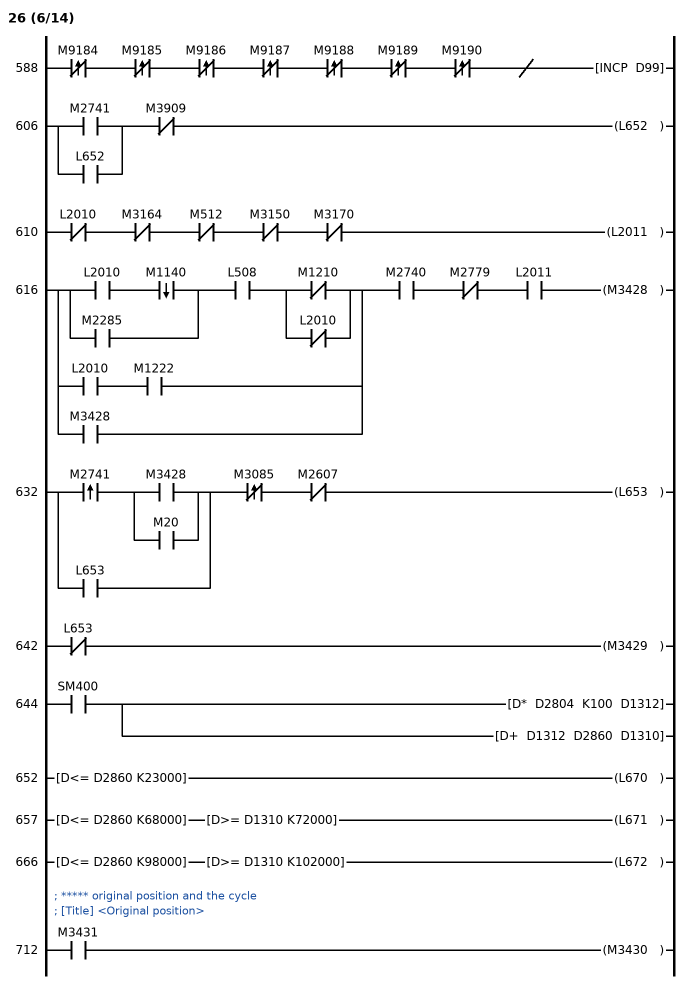
588   LDPI    M9184
      ANDPI   M9185
      ANDPI   M9186
      ANDPI   M9187
      ANDPI   M9188
      ANDPI   M9189
      ANDPI   M9190
      INV
      INCP    D99
606   LD      M2741
      OR      L652
      ANI     M3909
      OUT     L652
610   LDI     L2010
      ANI     M3164
      ANI     M512
      ANI     M3150
      ANI     M3170
      OUT     L2011
616   LD      L2010
      ANDF    M1140
      OR      M2285
      AND     L508
      LDI     M1210
      ORI     L2010
      ANB
      LD      L2010
      AND     M1222
      ORB
      OR      M3428
      AND     M2740
      ANI     M2779
      AND     L2011
      OUT     M3428
632   LDP     M2741
      LD      M3428
      OR      M20
      ANB
      OR      L653
      ANDPI   M3085
      ANI     M2607
      OUT     L653
642   LDI     L653
      OUT     M3429
644   LD      SM400
      D*      D2804 K100 D1312
      D+      D1312 D2860 D1310
652   LDD<=   D2860 K23000
      OUT     L670
657   LDD<=   D2860 K68000
      ANDD>=  D1310 K72000
      OUT     L671
666   LDD<=   D2860 K98000
      ANDD>=  D1310 K102000
      OUT     L672
; ***** original position and the cycle
; [Title] <Original position>
712   LD      M3431
      OUT     M3430
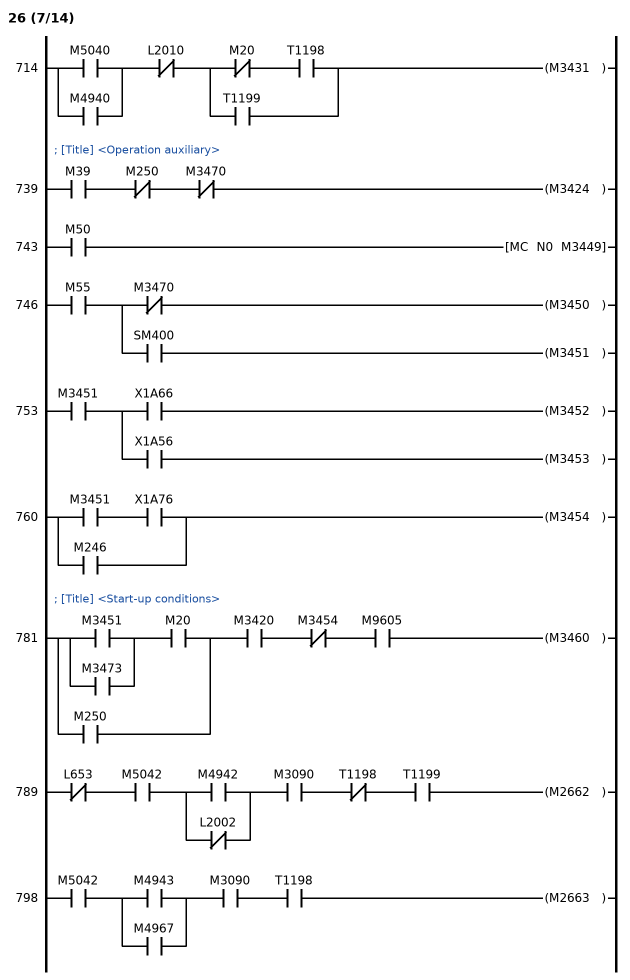
714   LD      M5040
      OR      M4940
      ANI     L2010
      LDI     M20
      AND     T1198
      OR      T1199
      ANB
      OUT     M3431
; [Title] <Operation auxiliary>
739   LD      M39
      ANI     M250
      ANI     M3470
      OUT     M3424
743   LD      M50
      MC      N0 M3449
746   LD      M55
      MPS
      ANI     M3470
      OUT     M3450
      MPP
      AND     SM400
      OUT     M3451
753   LD      M3451
      MPS
      AND     X1A66
      OUT     M3452
      MPP
      AND     X1A56
      OUT     M3453
760   LD      M3451
      AND     X1A76
      OR      M246
      OUT     M3454
; [Title] <Start-up conditions>
781   LD      M3451
      OR      M3473
      AND     M20
      OR      M250
      AND     M3420
      ANI     M3454
      AND     M9605
      OUT     M3460
789   LDI     L653
      AND     M5042
      LD      M4942
      ORI     L2002
      ANB
      AND     M3090
      ANI     T1198
      AND     T1199
      OUT     M2662
798   LD      M5042
      LD      M4943
      OR      M4967
      ANB
      AND     M3090
      AND     T1198
      OUT     M2663
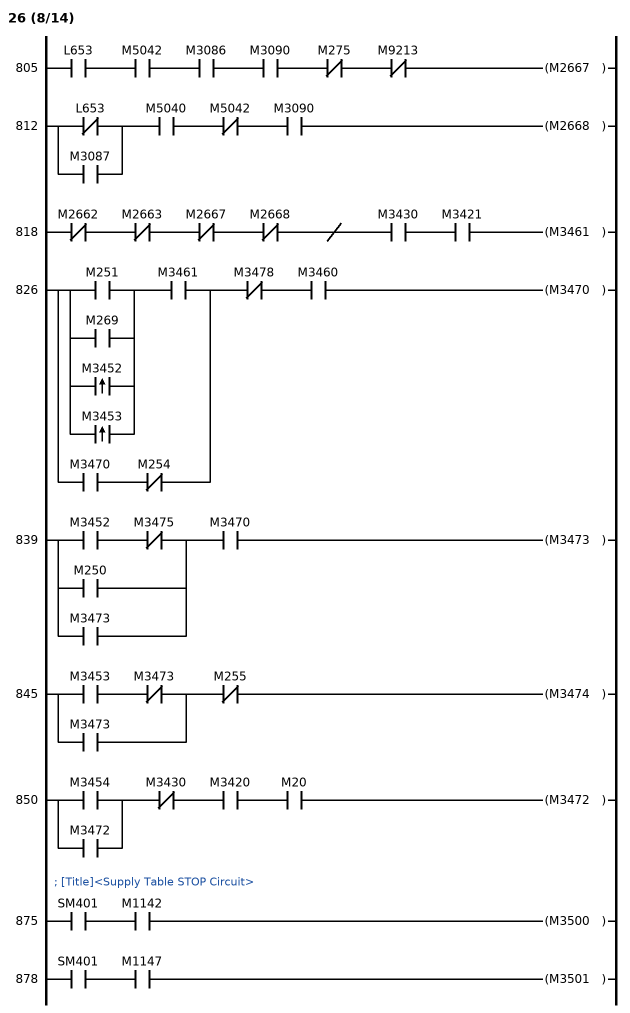
805   LD      L653
      AND     M5042
      AND     M3086
      AND     M3090
      ANI     M275
      ANI     M9213
      OUT     M2667
812   LDI     L653
      OR      M3087
      AND     M5040
      ANI     M5042
      AND     M3090
      OUT     M2668
818   LDI     M2662
      ANI     M2663
      ANI     M2667
      ANI     M2668
      INV
      AND     M3430
      AND     M3421
      OUT     M3461
826   LD      M251
      OR      M269
      ORP     M3452
      ORP     M3453
      AND     M3461
      LD      M3470
      ANI     M254
      ORB
      ANI     M3478
      AND     M3460
      OUT     M3470
839   LD      M3452
      ANI     M3475
      OR      M250
      OR      M3473
      AND     M3470
      OUT     M3473
845   LD      M3453
      ANI     M3473
      OR      M3473
      ANI     M255
      OUT     M3474
850   LD      M3454
      OR      M3472
      ANI     M3430
      AND     M3420
      AND     M20
      OUT     M3472
; [Title]<Supply Table STOP Circuit>
875   LD      SM401
      AND     M1142
      OUT     M3500
878   LD      SM401
      AND     M1147
      OUT     M3501
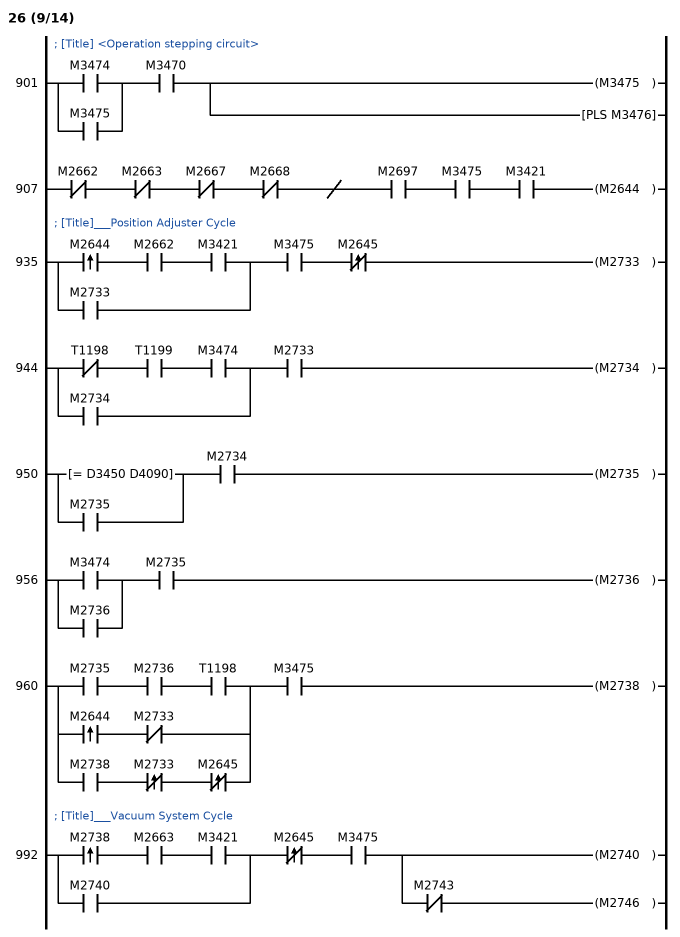
; [Title] <Operation stepping circuit>
901   LD      M3474
      OR      M3475
      AND     M3470
      OUT     M3475
      PLS     M3476
907   LDI     M2662
      ANI     M2663
      ANI     M2667
      ANI     M2668
      INV
      AND     M2697
      AND     M3475
      AND     M3421
      OUT     M2644
; [Title]___Position Adjuster Cycle
935   LDP     M2644
      AND     M2662
      AND     M3421
      OR      M2733
      AND     M3475
      ANDPI   M2645
      OUT     M2733
944   LDI     T1198
      AND     T1199
      AND     M3474
      OR      M2734
      AND     M2733
      OUT     M2734
950   LD=     D3450 D4090
      OR      M2735
      AND     M2734
      OUT     M2735
956   LD      M3474
      OR      M2736
      AND     M2735
      OUT     M2736
960   LD      M2735
      AND     M2736
      AND     T1198
      LDP     M2644
      ANI     M2733
      ORB
      LD      M2738
      ANDPI   M2733
      ANDPI   M2645
      ORB
      AND     M3475
      OUT     M2738
; [Title]___Vacuum System Cycle
992   LDP     M2738
      AND     M2663
      AND     M3421
      OR      M2740
      ANDPI   M2645
      AND     M3475
      OUT     M2740
      ANI     M2743
      OUT     M2746
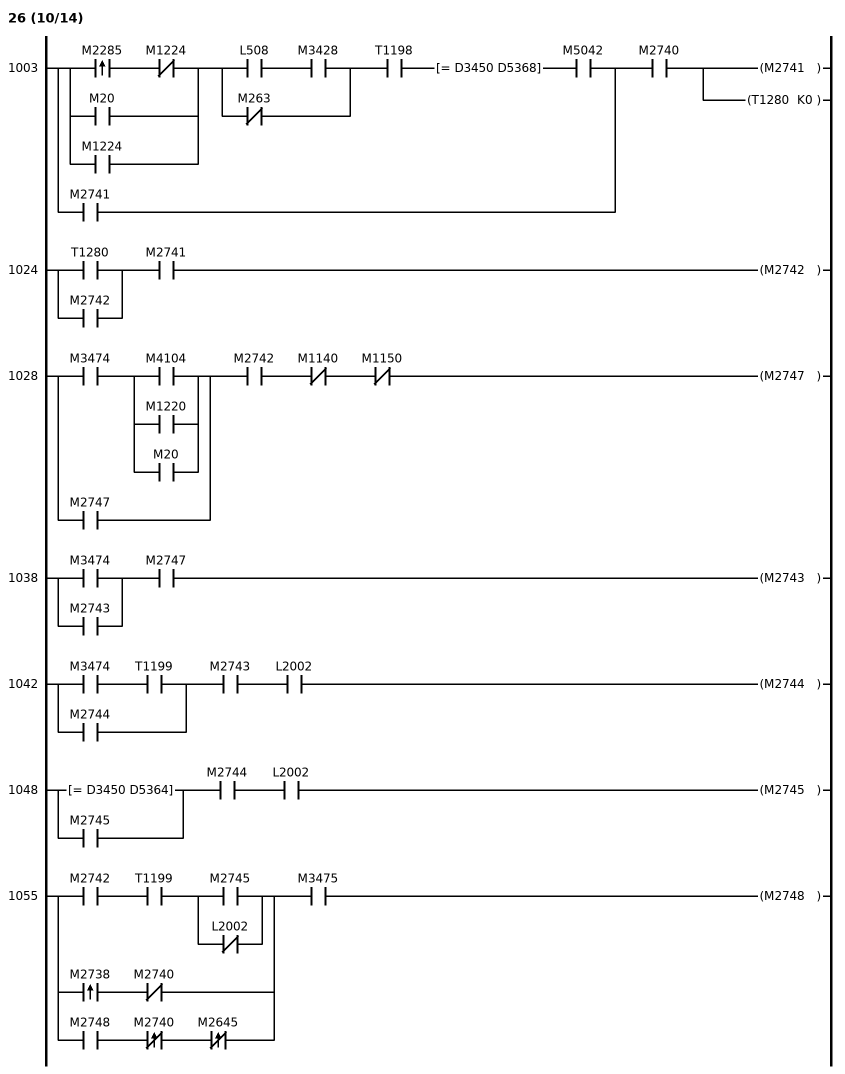
1003  LDP     M2285
      ANI     M1224
      OR      M20
      OR      M1224
      LD      L508
      AND     M3428
      ORI     M263
      ANB
      AND     T1198
      AND=    D3450 D5368
      AND     M5042
      OR      M2741
      AND     M2740
      OUT     M2741
      OUT     T1280 K0
1024  LD      T1280
      OR      M2742
      AND     M2741
      OUT     M2742
1028  LD      M3474
      LD      M4104
      OR      M1220
      OR      M20
      ANB
      OR      M2747
      AND     M2742
      ANI     M1140
      ANI     M1150
      OUT     M2747
1038  LD      M3474
      OR      M2743
      AND     M2747
      OUT     M2743
1042  LD      M3474
      AND     T1199
      OR      M2744
      AND     M2743
      AND     L2002
      OUT     M2744
1048  LD=     D3450 D5364
      OR      M2745
      AND     M2744
      AND     L2002
      OUT     M2745
1055  LD      M2742
      AND     T1199
      LD      M2745
      ORI     L2002
      ANB
      LDP     M2738
      ANI     M2740
      ORB
      LD      M2748
      ANDPI   M2740
      ANDPI   M2645
      ORB
      AND     M3475
      OUT     M2748
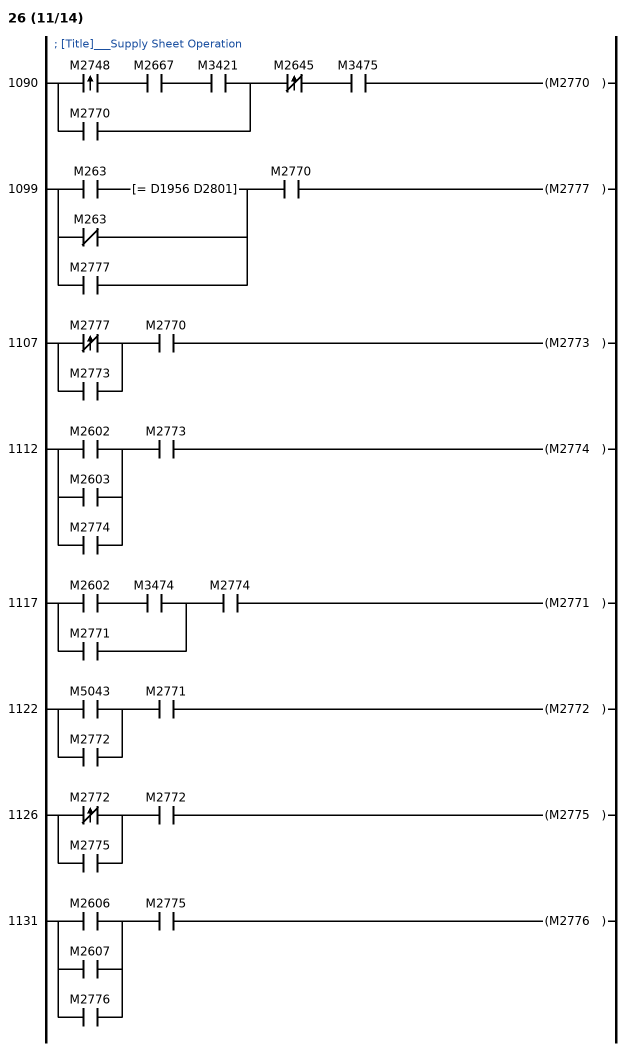
; [Title]___Supply Sheet Operation
1090  LDP     M2748
      AND     M2667
      AND     M3421
      OR      M2770
      ANDPI   M2645
      AND     M3475
      OUT     M2770
1099  LD      M263
      AND=    D1956 D2801
      ORI     M263
      OR      M2777
      AND     M2770
      OUT     M2777
1107  LDPI    M2777
      OR      M2773
      AND     M2770
      OUT     M2773
1112  LD      M2602
      OR      M2603
      OR      M2774
      AND     M2773
      OUT     M2774
1117  LD      M2602
      AND     M3474
      OR      M2771
      AND     M2774
      OUT     M2771
1122  LD      M5043
      OR      M2772
      AND     M2771
      OUT     M2772
1126  LDPI    M2772
      OR      M2775
      AND     M2772
      OUT     M2775
1131  LD      M2606
      OR      M2607
      OR      M2776
      AND     M2775
      OUT     M2776
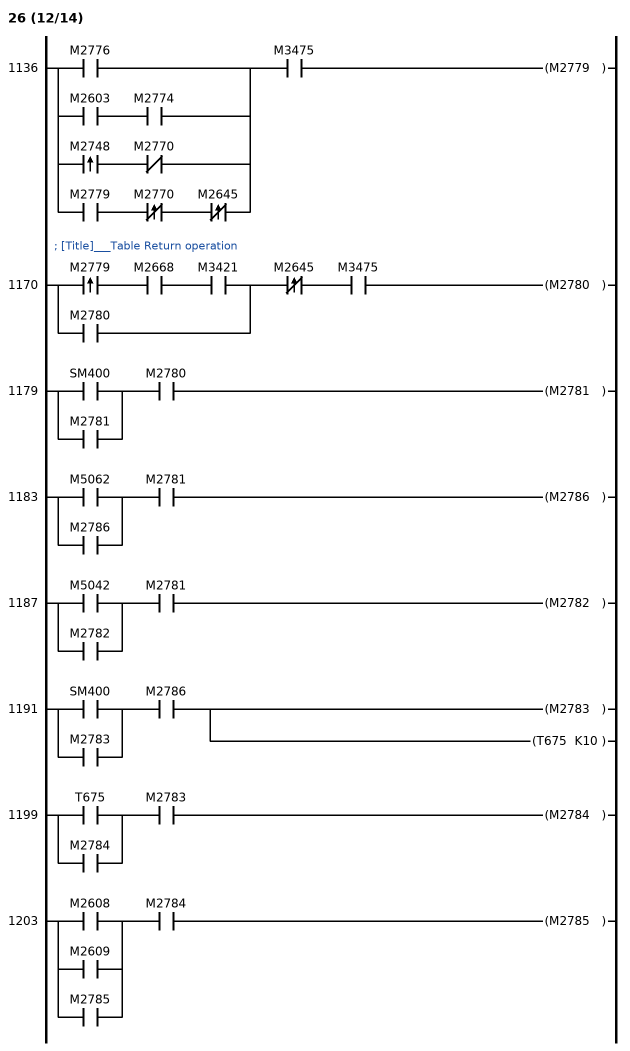
1136  LD      M2776
      LD      M2603
      AND     M2774
      ORB
      LDP     M2748
      ANI     M2770
      ORB
      LD      M2779
      ANDPI   M2770
      ANDPI   M2645
      ORB
      AND     M3475
      OUT     M2779
; [Title]___Table Return operation
1170  LDP     M2779
      AND     M2668
      AND     M3421
      OR      M2780
      ANDPI   M2645
      AND     M3475
      OUT     M2780
1179  LD      SM400
      OR      M2781
      AND     M2780
      OUT     M2781
1183  LD      M5062
      OR      M2786
      AND     M2781
      OUT     M2786
1187  LD      M5042
      OR      M2782
      AND     M2781
      OUT     M2782
1191  LD      SM400
      OR      M2783
      AND     M2786
      OUT     M2783
      OUT     T675 K10
1199  LD      T675
      OR      M2784
      AND     M2783
      OUT     M2784
1203  LD      M2608
      OR      M2609
      OR      M2785
      AND     M2784
      OUT     M2785
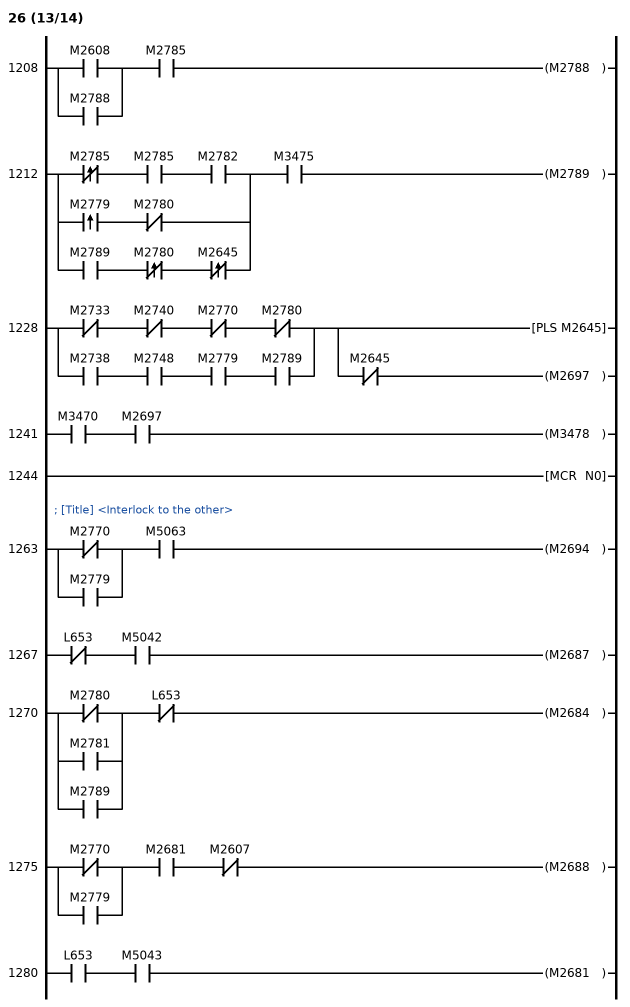
1208  LD      M2608
      OR      M2788
      AND     M2785
      OUT     M2788
1212  LDPI    M2785
      AND     M2785
      AND     M2782
      LDP     M2779
      ANI     M2780
      ORB
      LD      M2789
      ANDPI   M2780
      ANDPI   M2645
      ORB
      AND     M3475
      OUT     M2789
1228  LDI     M2733
      ANI     M2740
      ANI     M2770
      ANI     M2780
      LD      M2738
      AND     M2748
      AND     M2779
      AND     M2789
      ORB
      PLS     M2645
      ANI     M2645
      OUT     M2697
1241  LD      M3470
      AND     M2697
      OUT     M3478
1244  MCR     N0
; [Title] <Interlock to the other>
1263  LDI     M2770
      OR      M2779
      AND     M5063
      OUT     M2694
1267  LDI     L653
      AND     M5042
      OUT     M2687
1270  LDI     M2780
      OR      M2781
      OR      M2789
      ANI     L653
      OUT     M2684
1275  LDI     M2770
      OR      M2779
      AND     M2681
      ANI     M2607
      OUT     M2688
1280  LD      L653
      AND     M5043
      OUT     M2681
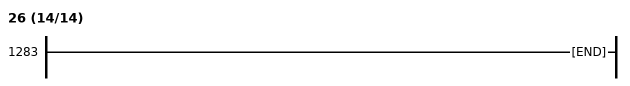
1283  END
END_PROGRAM

PROGRAM 70
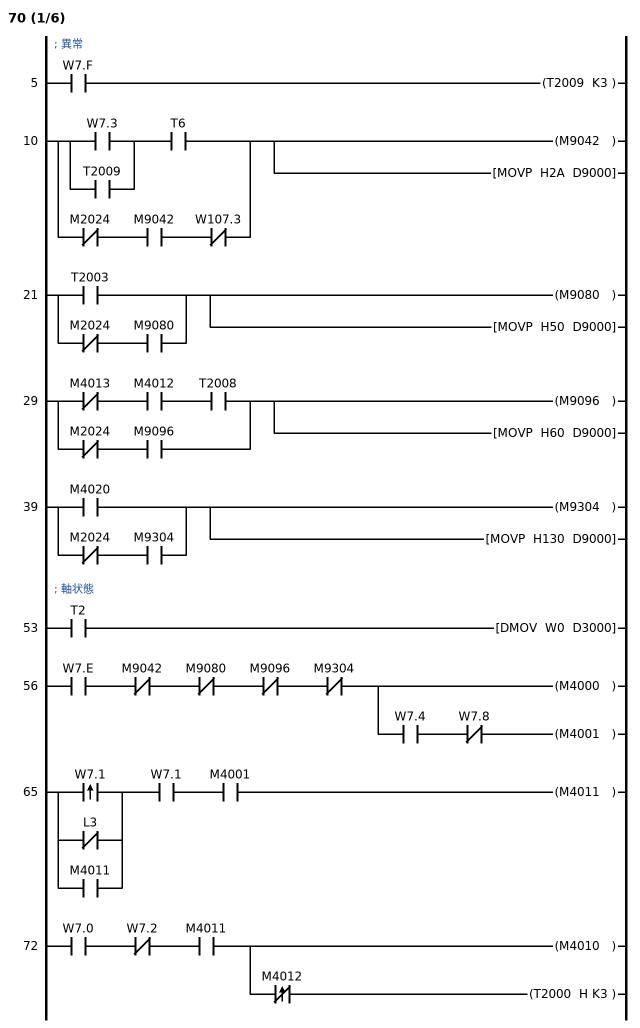
; 異常
5     LD      W7.F
      OUT     T2009 K3
10    LD      W7.3
      OR      T2009
      AND     T6
      LDI     M2024
      AND     M9042
      ANI     W107.3
      ORB
      OUT     M9042
      MOVP    H2A D9000
21    LD      T2003
      LDI     M2024
      AND     M9080
      ORB
      OUT     M9080
      MOVP    H50 D9000
29    LDI     M4013
      AND     M4012
      AND     T2008
      LDI     M2024
      AND     M9096
      ORB
      OUT     M9096
      MOVP    H60 D9000
39    LD      M4020
      LDI     M2024
      AND     M9304
      ORB
      OUT     M9304
      MOVP    H130 D9000
; 軸状態
53    LD      T2
      DMOV    W0 D3000
56    LD      W7.E
      ANI     M9042
      ANI     M9080
      ANI     M9096
      ANI     M9304
      OUT     M4000
      AND     W7.4
      ANI     W7.8
      OUT     M4001
65    LDP     W7.1
      ORI     L3
      OR      M4011
      AND     W7.1
      AND     M4001
      OUT     M4011
72    LD      W7.0
      ANI     W7.2
      AND     M4011
      OUT     M4010
      ANDPI   M4012
      OUTH    T2000 K3
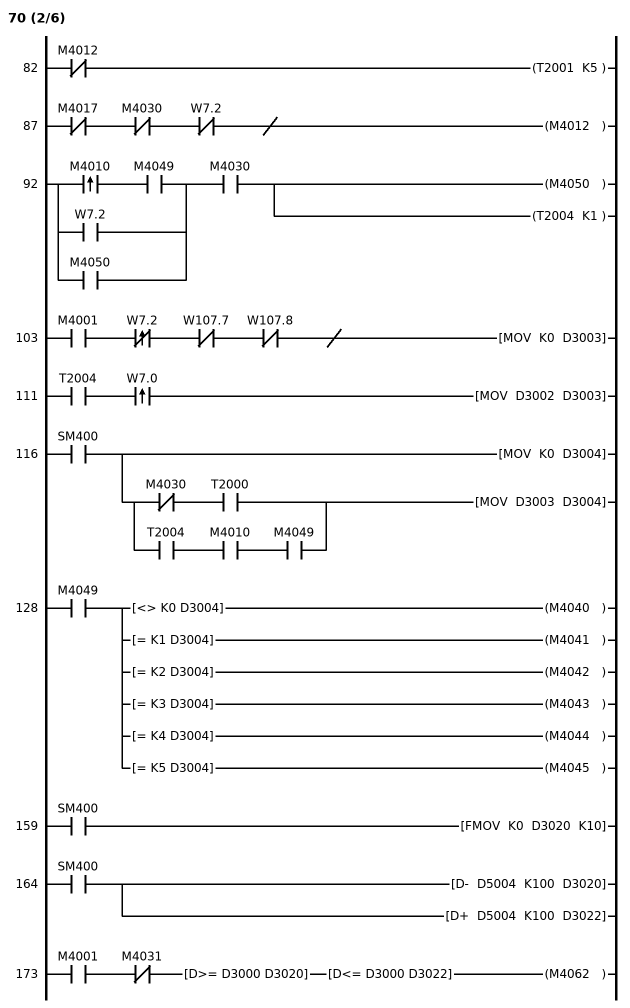
82    LDI     M4012
      OUT     T2001 K5
87    LDI     M4017
      ANI     M4030
      ANI     W7.2
      INV
      OUT     M4012
92    LDP     M4010
      AND     M4049
      OR      W7.2
      OR      M4050
      AND     M4030
      OUT     M4050
      OUT     T2004 K1
103   LD      M4001
      ANDPI   W7.2
      ANI     W107.7
      ANI     W107.8
      INV
      MOV     K0 D3003
111   LD      T2004
      ANDP    W7.0
      MOV     D3002 D3003
116   LD      SM400
      MOV     K0 D3004
      LDI     M4030
      AND     T2000
      LD      T2004
      AND     M4010
      AND     M4049
      ORB
      ANB
      MOV     D3003 D3004
128   LD      M4049
      MPS
      AND<>   K0 D3004
      OUT     M4040
      MRD
      AND=    K1 D3004
      OUT     M4041
      MRD
      AND=    K2 D3004
      OUT     M4042
      MRD
      AND=    K3 D3004
      OUT     M4043
      MRD
      AND=    K4 D3004
      OUT     M4044
      MPP
      AND=    K5 D3004
      OUT     M4045
159   LD      SM400
      FMOV    K0 D3020 K10
164   LD      SM400
      D-      D5004 K100 D3020
      D+      D5004 K100 D3022
173   LD      M4001
      ANI     M4031
      ANDD>=  D3000 D3020
      ANDD<=  D3000 D3022
      OUT     M4062
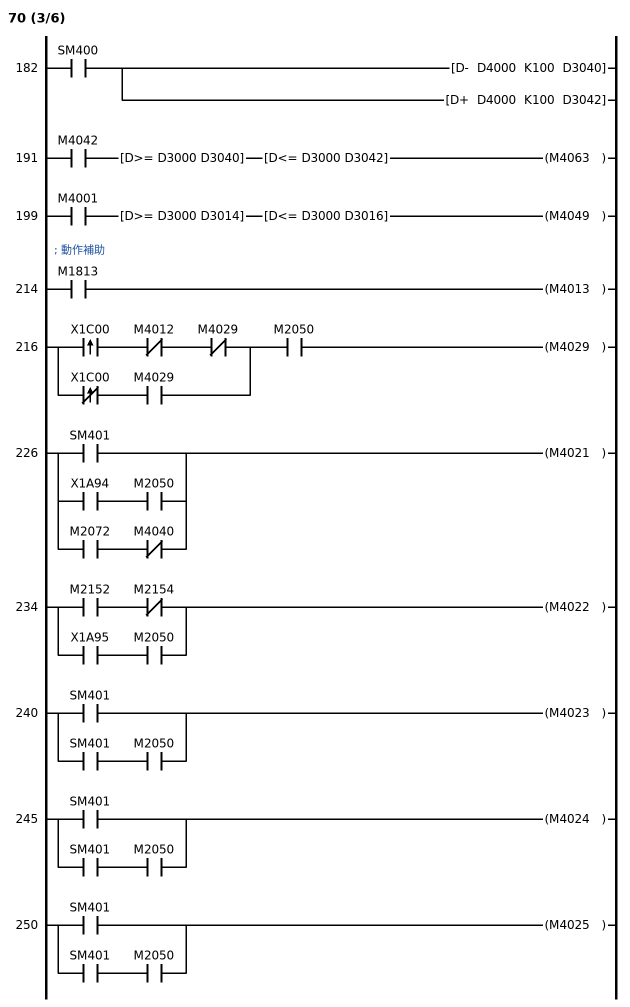
182   LD      SM400
      D-      D4000 K100 D3040
      D+      D4000 K100 D3042
191   LD      M4042
      ANDD>=  D3000 D3040
      ANDD<=  D3000 D3042
      OUT     M4063
199   LD      M4001
      ANDD>=  D3000 D3014
      ANDD<=  D3000 D3016
      OUT     M4049
; 動作補助
214   LD      M1813
      OUT     M4013
216   LDP     X1C00
      ANI     M4012
      ANI     M4029
      LDPI    X1C00
      AND     M4029
      ORB
      AND     M2050
      OUT     M4029
226   LD      SM401
      LD      X1A94
      AND     M2050
      ORB
      LD      M2072
      ANI     M4040
      ORB
      OUT     M4021
234   LD      M2152
      ANI     M2154
      LD      X1A95
      AND     M2050
      ORB
      OUT     M4022
240   LD      SM401
      LD      SM401
      AND     M2050
      ORB
      OUT     M4023
245   LD      SM401
      LD      SM401
      AND     M2050
      ORB
      OUT     M4024
250   LD      SM401
      LD      SM401
      AND     M2050
      ORB
      OUT     M4025
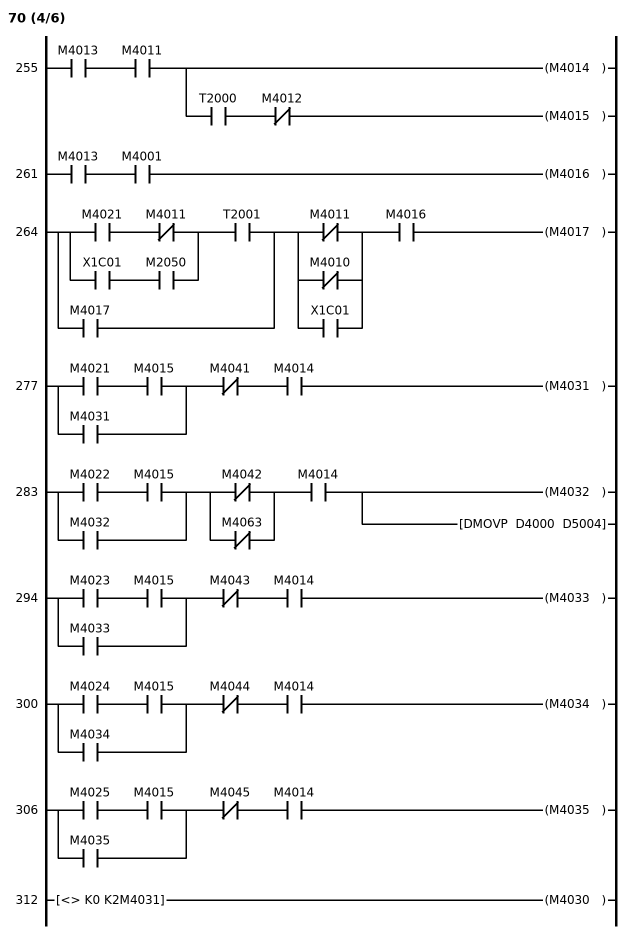
255   LD      M4013
      AND     M4011
      OUT     M4014
      AND     T2000
      ANI     M4012
      OUT     M4015
261   LD      M4013
      AND     M4001
      OUT     M4016
264   LD      M4021
      ANI     M4011
      LD      X1C01
      AND     M2050
      ORB
      AND     T2001
      OR      M4017
      LDI     M4011
      ORI     M4010
      OR      X1C01
      ANB
      AND     M4016
      OUT     M4017
277   LD      M4021
      AND     M4015
      OR      M4031
      ANI     M4041
      AND     M4014
      OUT     M4031
283   LD      M4022
      AND     M4015
      OR      M4032
      LDI     M4042
      ORI     M4063
      ANB
      AND     M4014
      OUT     M4032
      DMOVP   D4000 D5004
294   LD      M4023
      AND     M4015
      OR      M4033
      ANI     M4043
      AND     M4014
      OUT     M4033
300   LD      M4024
      AND     M4015
      OR      M4034
      ANI     M4044
      AND     M4014
      OUT     M4034
306   LD      M4025
      AND     M4015
      OR      M4035
      ANI     M4045
      AND     M4014
      OUT     M4035
312   LD<>    K0 K2M4031
      OUT     M4030
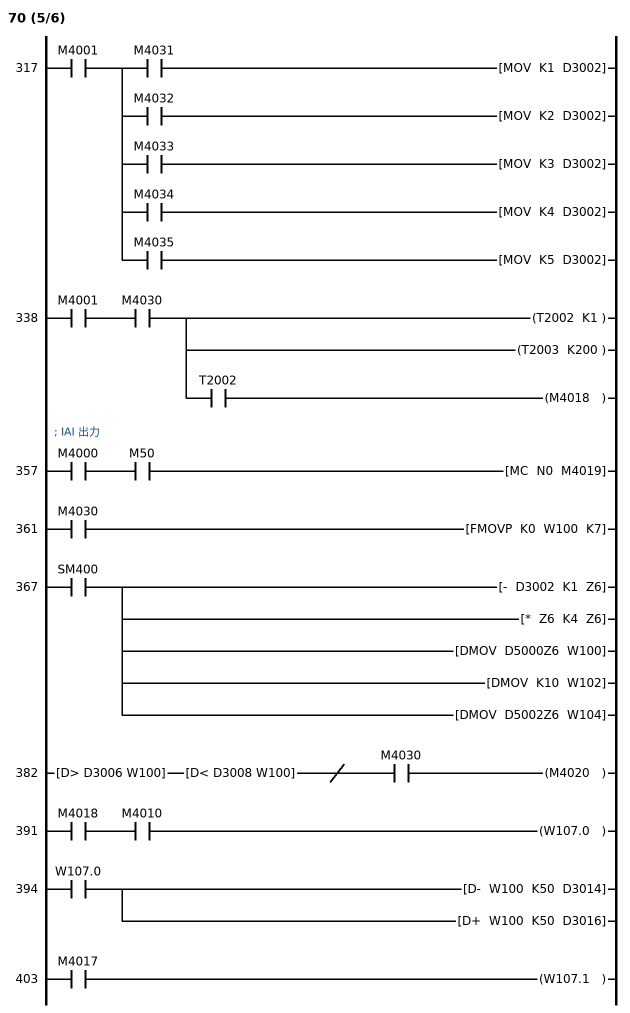
317   LD      M4001
      MPS
      AND     M4031
      MOV     K1 D3002
      MRD
      AND     M4032
      MOV     K2 D3002
      MRD
      AND     M4033
      MOV     K3 D3002
      MRD
      AND     M4034
      MOV     K4 D3002
      MPP
      AND     M4035
      MOV     K5 D3002
338   LD      M4001
      AND     M4030
      OUT     T2002 K1
      OUT     T2003 K200
      AND     T2002
      OUT     M4018
; IAI 出力
357   LD      M4000
      AND     M50
      MC      N0 M4019
361   LD      M4030
      FMOVP   K0 W100 K7
367   LD      SM400
      -       D3002 K1 Z6
      *       Z6 K4 Z6
      DMOV    D5000Z6 W100
      DMOV    K10 W102
      DMOV    D5002Z6 W104
382   LDD>    D3006 W100
      ANDD<   D3008 W100
      INV
      AND     M4030
      OUT     M4020
391   LD      M4018
      AND     M4010
      OUT     W107.0
394   LD      W107.0
      D-      W100 K50 D3014
      D+      W100 K50 D3016
403   LD      M4017
      OUT     W107.1
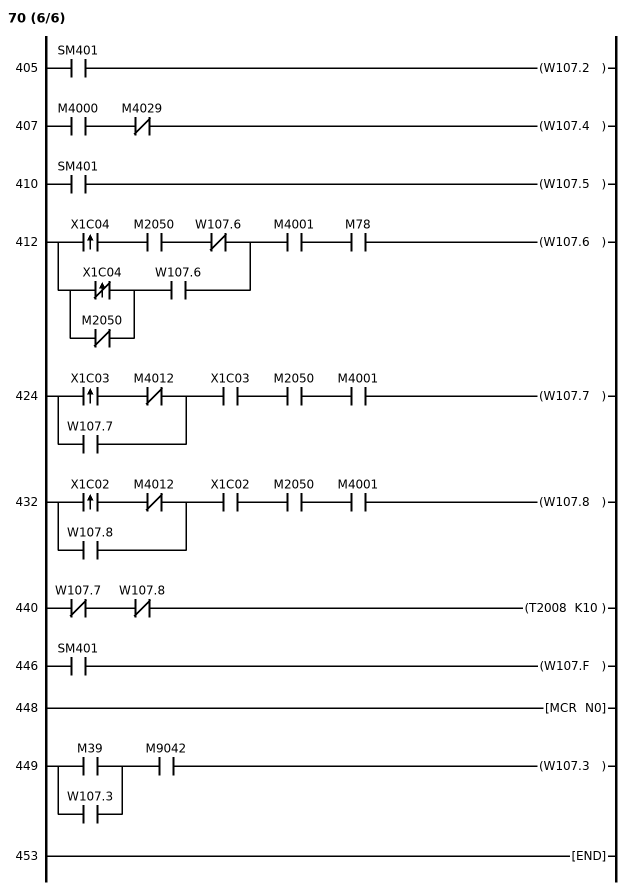
405   LD      SM401
      OUT     W107.2
407   LD      M4000
      ANI     M4029
      OUT     W107.4
410   LD      SM401
      OUT     W107.5
412   LDP     X1C04
      AND     M2050
      ANI     W107.6
      LDPI    X1C04
      ORI     M2050
      AND     W107.6
      ORB
      AND     M4001
      AND     M78
      OUT     W107.6
424   LDP     X1C03
      ANI     M4012
      OR      W107.7
      AND     X1C03
      AND     M2050
      AND     M4001
      OUT     W107.7
432   LDP     X1C02
      ANI     M4012
      OR      W107.8
      AND     X1C02
      AND     M2050
      AND     M4001
      OUT     W107.8
440   LDI     W107.7
      ANI     W107.8
      OUT     T2008 K10
446   LD      SM401
      OUT     W107.F
448   MCR     N0
449   LD      M39
      OR      W107.3
      AND     M9042
      OUT     W107.3
453   END
END_PROGRAM

PROGRAM 71
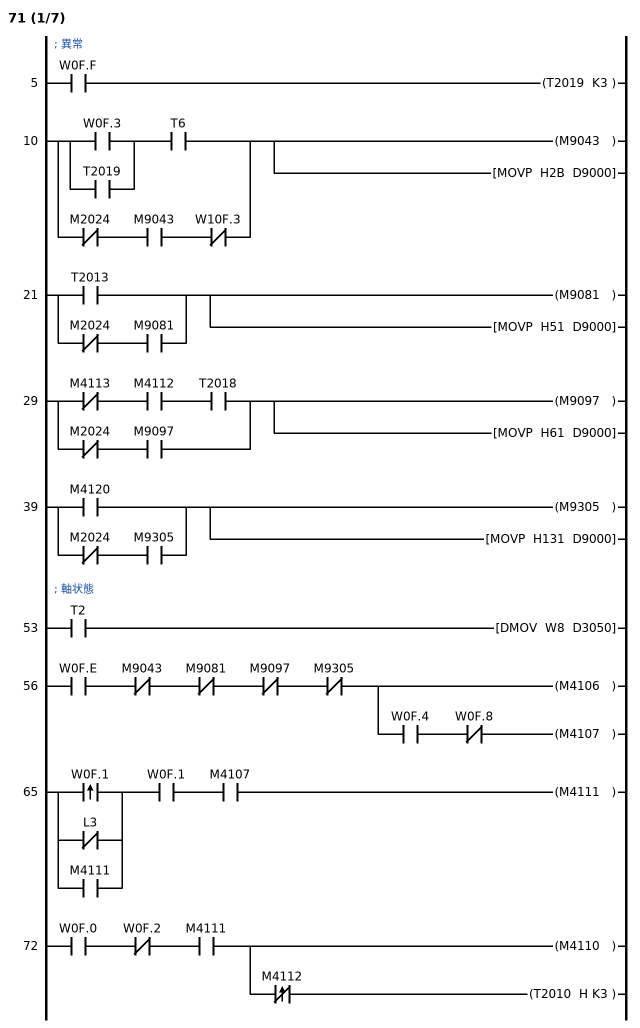
; 異常
5     LD      W0F.F
      OUT     T2019 K3
10    LD      W0F.3
      OR      T2019
      AND     T6
      LDI     M2024
      AND     M9043
      ANI     W10F.3
      ORB
      OUT     M9043
      MOVP    H2B D9000
21    LD      T2013
      LDI     M2024
      AND     M9081
      ORB
      OUT     M9081
      MOVP    H51 D9000
29    LDI     M4113
      AND     M4112
      AND     T2018
      LDI     M2024
      AND     M9097
      ORB
      OUT     M9097
      MOVP    H61 D9000
39    LD      M4120
      LDI     M2024
      AND     M9305
      ORB
      OUT     M9305
      MOVP    H131 D9000
; 軸状態
53    LD      T2
      DMOV    W8 D3050
56    LD      W0F.E
      ANI     M9043
      ANI     M9081
      ANI     M9097
      ANI     M9305
      OUT     M4106
      AND     W0F.4
      ANI     W0F.8
      OUT     M4107
65    LDP     W0F.1
      ORI     L3
      OR      M4111
      AND     W0F.1
      AND     M4107
      OUT     M4111
72    LD      W0F.0
      ANI     W0F.2
      AND     M4111
      OUT     M4110
      ANDPI   M4112
      OUTH    T2010 K3
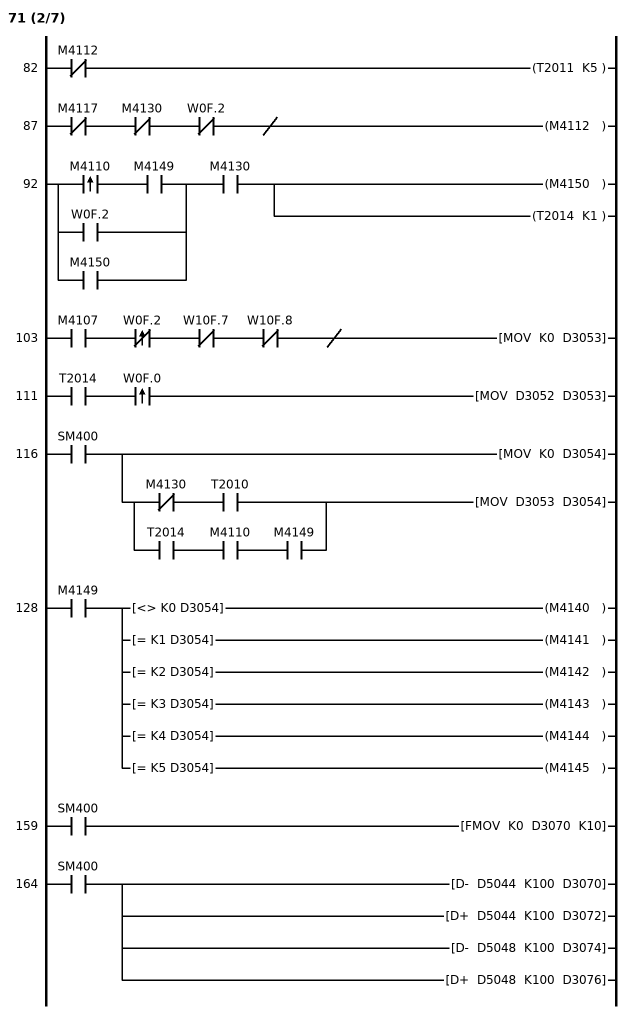
82    LDI     M4112
      OUT     T2011 K5
87    LDI     M4117
      ANI     M4130
      ANI     W0F.2
      INV
      OUT     M4112
92    LDP     M4110
      AND     M4149
      OR      W0F.2
      OR      M4150
      AND     M4130
      OUT     M4150
      OUT     T2014 K1
103   LD      M4107
      ANDPI   W0F.2
      ANI     W10F.7
      ANI     W10F.8
      INV
      MOV     K0 D3053
111   LD      T2014
      ANDP    W0F.0
      MOV     D3052 D3053
116   LD      SM400
      MOV     K0 D3054
      LDI     M4130
      AND     T2010
      LD      T2014
      AND     M4110
      AND     M4149
      ORB
      ANB
      MOV     D3053 D3054
128   LD      M4149
      MPS
      AND<>   K0 D3054
      OUT     M4140
      MRD
      AND=    K1 D3054
      OUT     M4141
      MRD
      AND=    K2 D3054
      OUT     M4142
      MRD
      AND=    K3 D3054
      OUT     M4143
      MRD
      AND=    K4 D3054
      OUT     M4144
      MPP
      AND=    K5 D3054
      OUT     M4145
159   LD      SM400
      FMOV    K0 D3070 K10
164   LD      SM400
      D-      D5044 K100 D3070
      D+      D5044 K100 D3072
      D-      D5048 K100 D3074
      D+      D5048 K100 D3076
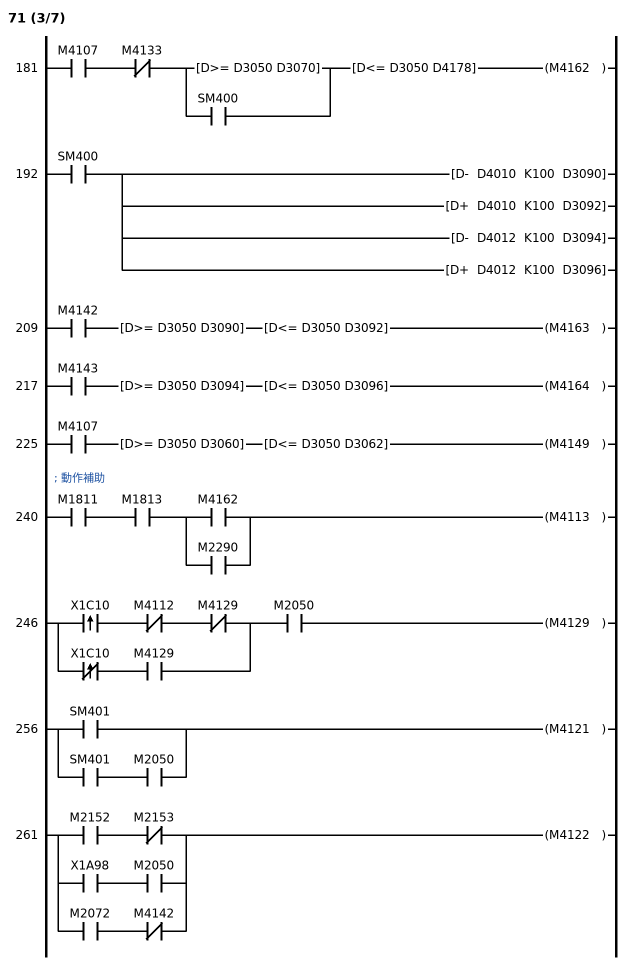
181   LD      M4107
      ANI     M4133
      LDD>=   D3050 D3070
      OR      SM400
      ANB
      ANDD<=  D3050 D4178
      OUT     M4162
192   LD      SM400
      D-      D4010 K100 D3090
      D+      D4010 K100 D3092
      D-      D4012 K100 D3094
      D+      D4012 K100 D3096
209   LD      M4142
      ANDD>=  D3050 D3090
      ANDD<=  D3050 D3092
      OUT     M4163
217   LD      M4143
      ANDD>=  D3050 D3094
      ANDD<=  D3050 D3096
      OUT     M4164
225   LD      M4107
      ANDD>=  D3050 D3060
      ANDD<=  D3050 D3062
      OUT     M4149
; 動作補助
240   LD      M1811
      AND     M1813
      LD      M4162
      OR      M2290
      ANB
      OUT     M4113
246   LDP     X1C10
      ANI     M4112
      ANI     M4129
      LDPI    X1C10
      AND     M4129
      ORB
      AND     M2050
      OUT     M4129
256   LD      SM401
      LD      SM401
      AND     M2050
      ORB
      OUT     M4121
261   LD      M2152
      ANI     M2153
      LD      X1A98
      AND     M2050
      ORB
      LD      M2072
      ANI     M4142
      ORB
      OUT     M4122
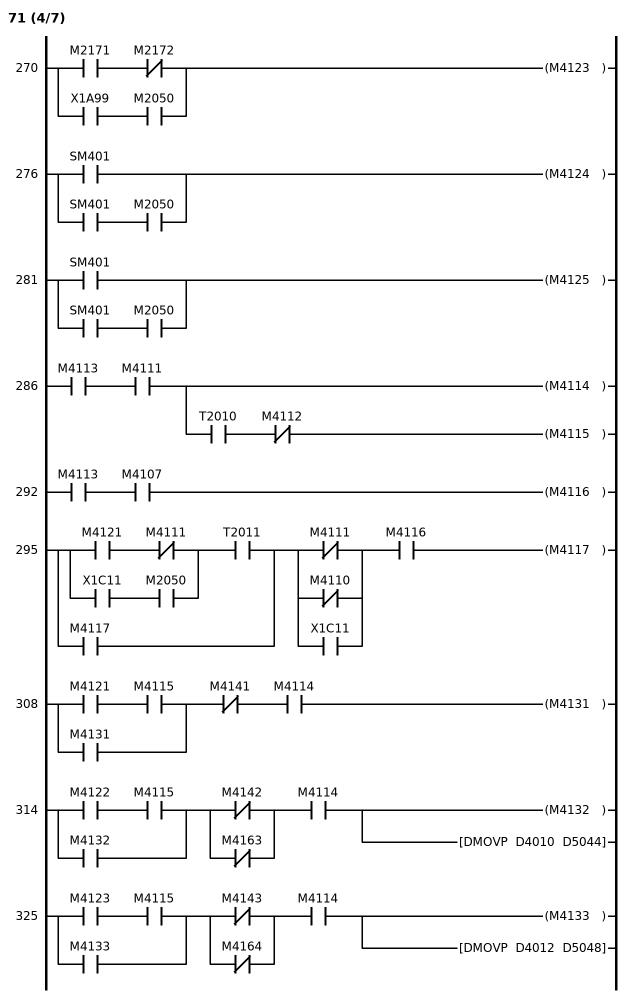
270   LD      M2171
      ANI     M2172
      LD      X1A99
      AND     M2050
      ORB
      OUT     M4123
276   LD      SM401
      LD      SM401
      AND     M2050
      ORB
      OUT     M4124
281   LD      SM401
      LD      SM401
      AND     M2050
      ORB
      OUT     M4125
286   LD      M4113
      AND     M4111
      OUT     M4114
      AND     T2010
      ANI     M4112
      OUT     M4115
292   LD      M4113
      AND     M4107
      OUT     M4116
295   LD      M4121
      ANI     M4111
      LD      X1C11
      AND     M2050
      ORB
      AND     T2011
      OR      M4117
      LDI     M4111
      ORI     M4110
      OR      X1C11
      ANB
      AND     M4116
      OUT     M4117
308   LD      M4121
      AND     M4115
      OR      M4131
      ANI     M4141
      AND     M4114
      OUT     M4131
314   LD      M4122
      AND     M4115
      OR      M4132
      LDI     M4142
      ORI     M4163
      ANB
      AND     M4114
      OUT     M4132
      DMOVP   D4010 D5044
325   LD      M4123
      AND     M4115
      OR      M4133
      LDI     M4143
      ORI     M4164
      ANB
      AND     M4114
      OUT     M4133
      DMOVP   D4012 D5048
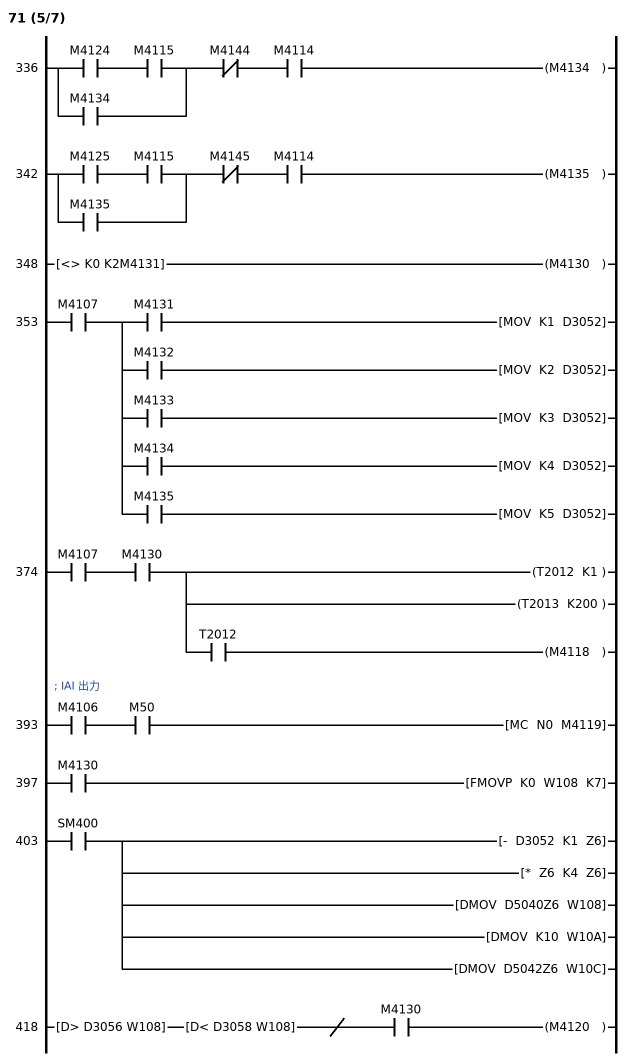
336   LD      M4124
      AND     M4115
      OR      M4134
      ANI     M4144
      AND     M4114
      OUT     M4134
342   LD      M4125
      AND     M4115
      OR      M4135
      ANI     M4145
      AND     M4114
      OUT     M4135
348   LD<>    K0 K2M4131
      OUT     M4130
353   LD      M4107
      MPS
      AND     M4131
      MOV     K1 D3052
      MRD
      AND     M4132
      MOV     K2 D3052
      MRD
      AND     M4133
      MOV     K3 D3052
      MRD
      AND     M4134
      MOV     K4 D3052
      MPP
      AND     M4135
      MOV     K5 D3052
374   LD      M4107
      AND     M4130
      OUT     T2012 K1
      OUT     T2013 K200
      AND     T2012
      OUT     M4118
; IAI 出力
393   LD      M4106
      AND     M50
      MC      N0 M4119
397   LD      M4130
      FMOVP   K0 W108 K7
403   LD      SM400
      -       D3052 K1 Z6
      *       Z6 K4 Z6
      DMOV    D5040Z6 W108
      DMOV    K10 W10A
      DMOV    D5042Z6 W10C
418   LDD>    D3056 W108
      ANDD<   D3058 W108
      INV
      AND     M4130
      OUT     M4120
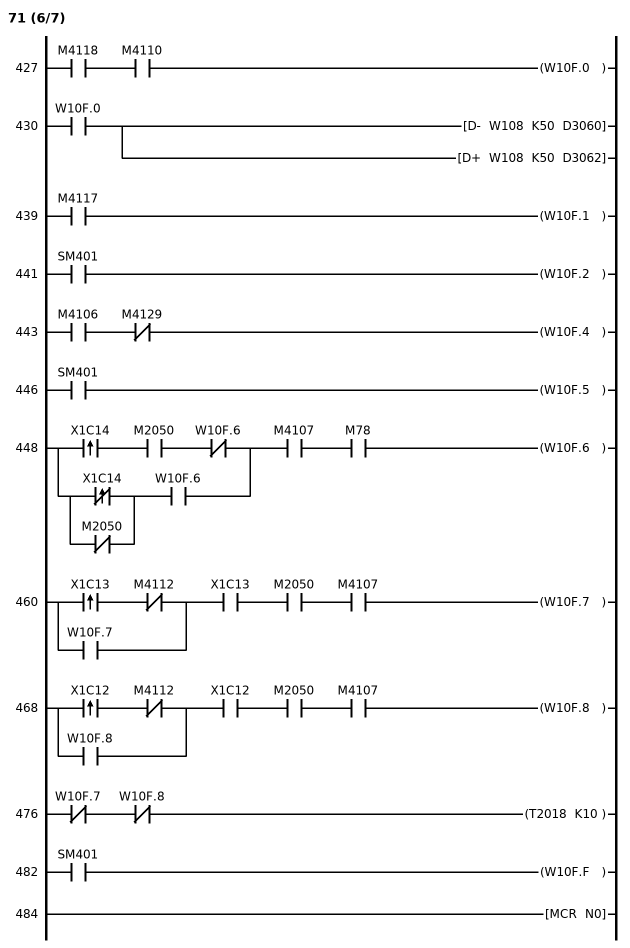
427   LD      M4118
      AND     M4110
      OUT     W10F.0
430   LD      W10F.0
      D-      W108 K50 D3060
      D+      W108 K50 D3062
439   LD      M4117
      OUT     W10F.1
441   LD      SM401
      OUT     W10F.2
443   LD      M4106
      ANI     M4129
      OUT     W10F.4
446   LD      SM401
      OUT     W10F.5
448   LDP     X1C14
      AND     M2050
      ANI     W10F.6
      LDPI    X1C14
      ORI     M2050
      AND     W10F.6
      ORB
      AND     M4107
      AND     M78
      OUT     W10F.6
460   LDP     X1C13
      ANI     M4112
      OR      W10F.7
      AND     X1C13
      AND     M2050
      AND     M4107
      OUT     W10F.7
468   LDP     X1C12
      ANI     M4112
      OR      W10F.8
      AND     X1C12
      AND     M2050
      AND     M4107
      OUT     W10F.8
476   LDI     W10F.7
      ANI     W10F.8
      OUT     T2018 K10
482   LD      SM401
      OUT     W10F.F
484   MCR     N0
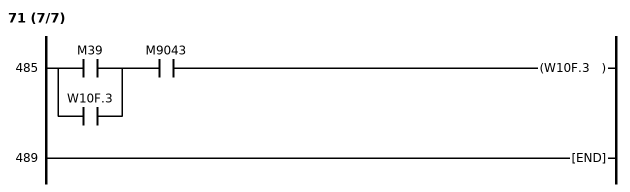
485   LD      M39
      OR      W10F.3
      AND     M9043
      OUT     W10F.3
489   END
END_PROGRAM

PROGRAM 72
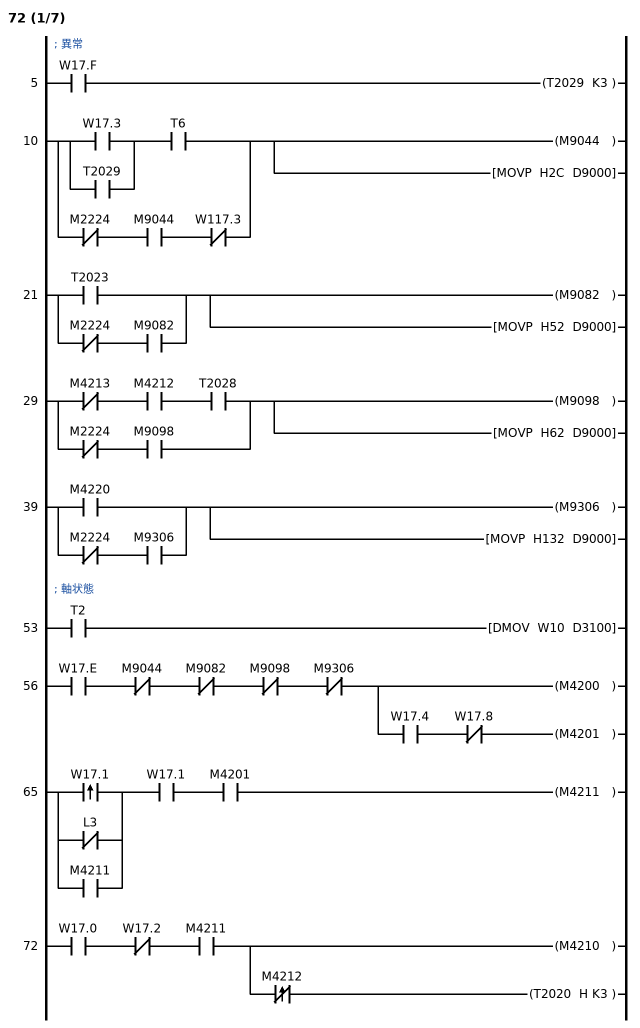
; 異常
5     LD      W17.F
      OUT     T2029 K3
10    LD      W17.3
      OR      T2029
      AND     T6
      LDI     M2224
      AND     M9044
      ANI     W117.3
      ORB
      OUT     M9044
      MOVP    H2C D9000
21    LD      T2023
      LDI     M2224
      AND     M9082
      ORB
      OUT     M9082
      MOVP    H52 D9000
29    LDI     M4213
      AND     M4212
      AND     T2028
      LDI     M2224
      AND     M9098
      ORB
      OUT     M9098
      MOVP    H62 D9000
39    LD      M4220
      LDI     M2224
      AND     M9306
      ORB
      OUT     M9306
      MOVP    H132 D9000
; 軸状態
53    LD      T2
      DMOV    W10 D3100
56    LD      W17.E
      ANI     M9044
      ANI     M9082
      ANI     M9098
      ANI     M9306
      OUT     M4200
      AND     W17.4
      ANI     W17.8
      OUT     M4201
65    LDP     W17.1
      ORI     L3
      OR      M4211
      AND     W17.1
      AND     M4201
      OUT     M4211
72    LD      W17.0
      ANI     W17.2
      AND     M4211
      OUT     M4210
      ANDPI   M4212
      OUTH    T2020 K3
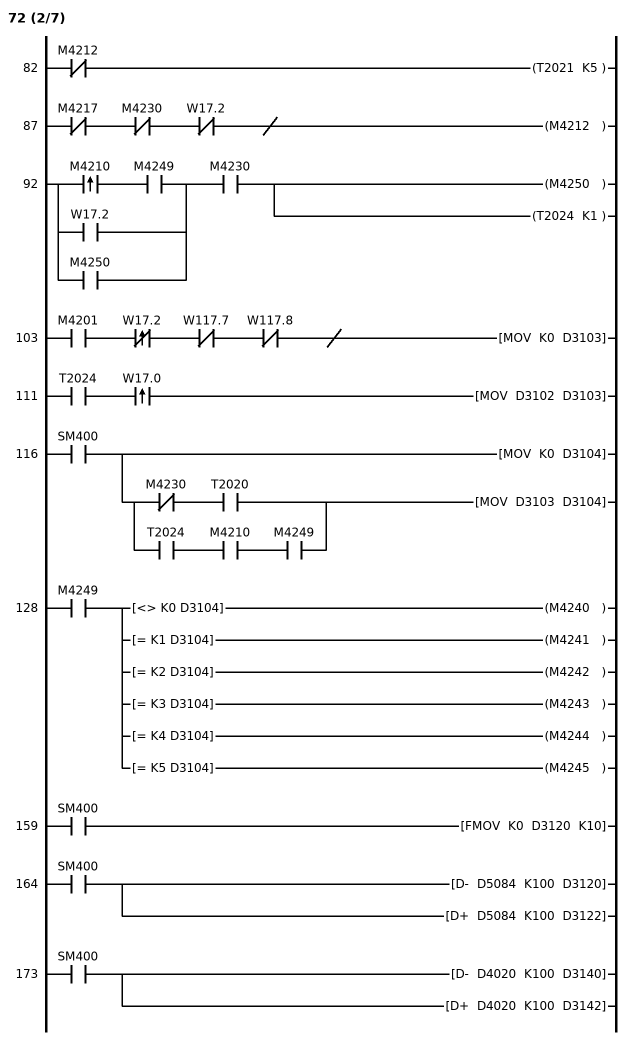
82    LDI     M4212
      OUT     T2021 K5
87    LDI     M4217
      ANI     M4230
      ANI     W17.2
      INV
      OUT     M4212
92    LDP     M4210
      AND     M4249
      OR      W17.2
      OR      M4250
      AND     M4230
      OUT     M4250
      OUT     T2024 K1
103   LD      M4201
      ANDPI   W17.2
      ANI     W117.7
      ANI     W117.8
      INV
      MOV     K0 D3103
111   LD      T2024
      ANDP    W17.0
      MOV     D3102 D3103
116   LD      SM400
      MOV     K0 D3104
      LDI     M4230
      AND     T2020
      LD      T2024
      AND     M4210
      AND     M4249
      ORB
      ANB
      MOV     D3103 D3104
128   LD      M4249
      MPS
      AND<>   K0 D3104
      OUT     M4240
      MRD
      AND=    K1 D3104
      OUT     M4241
      MRD
      AND=    K2 D3104
      OUT     M4242
      MRD
      AND=    K3 D3104
      OUT     M4243
      MRD
      AND=    K4 D3104
      OUT     M4244
      MPP
      AND=    K5 D3104
      OUT     M4245
159   LD      SM400
      FMOV    K0 D3120 K10
164   LD      SM400
      D-      D5084 K100 D3120
      D+      D5084 K100 D3122
173   LD      SM400
      D-      D4020 K100 D3140
      D+      D4020 K100 D3142
